{attribute 'GeneratedUsingTerminal: EM7004-0000-9995'}
{attribute addProperty BoxType "EM7004-0000-9995"}
{attribute addProperty Id "OutputAT %Q*INT2"}
{attribute addProperty CRC "1604026022"}
{attribute addProperty Size "2"}
TYPE Analog_Channel_5F9B7EA6 :
STRUCT
	{attribute addProperty Name "Output"}
	Output AT %Q* : INT;
END_STRUCT
END_TYPE

(* stored: Version 1.2.0.0, ProductVersion 3.1.4024.9
   DUT Analog_Channel_5F9B7EA6: Id {5e65735a-5d19-4085-8108-553edf4f78dc} *)
